KUKA KRL program: makrosaw.src

&ACCESS RV
&PARAM TEMPLATE = C:\KRC\Roboter\Template\makrosawvorgabe.src
&PARAM EDITMASK = MakroSAW
&PARAM TPVW_VERSION=8.3.17
DEF  MAKROSAW ( )
; FOLD Makro Anfang;%{PSE} %MKUKATPVW
SPS_N=-1
; ENDFOLD
; FOLD ;%{H}
END
; ENDFOLD
